FUNCTION_BLOCK FB_SFC_SamplePou
VAR_INPUT
//	eOperation	: INT;
	eOperation	: E_Operation;
END_VAR
VAR_OUTPUT
	iResultC	: DINT;
END_VAR
VAR
	arrDataA	: ARRAY [1..iMax] OF DINT;
	arrDataB	: ARRAY [1..iMax] OF DINT;
	arrDataC	: ARRAY [1..iMax] OF DINT;
	I 			: DINT;
	bInit		: BOOL := TRUE;
	bAdd		: BOOL;
	bSub		: BOOL;
	bMul		: BOOL;
END_VAR
VAR CONSTANT
	iMax 		: DINT := 10;
END_VAR

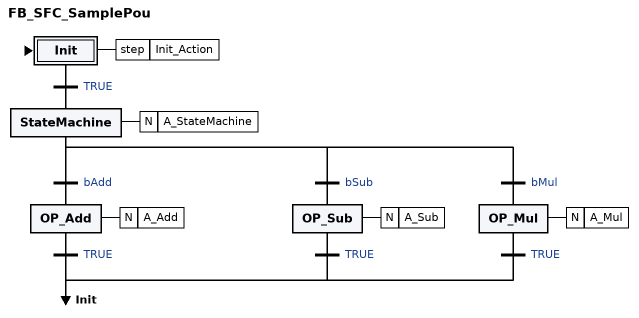
INITIAL_STEP Init:
    Init_Action(N);  // step action
END_STEP
TRANSITION FROM Init TO StateMachine
    := TRUE;
END_TRANSITION
STEP StateMachine:
    A_StateMachine(N);
END_STEP
TRANSITION FROM StateMachine TO OP_Add
    := bAdd;
END_TRANSITION
STEP OP_Add:
    A_Add(N);
END_STEP
TRANSITION FROM OP_Add TO Init
    := TRUE;
END_TRANSITION
TRANSITION FROM StateMachine TO OP_Sub
    := bSub;
END_TRANSITION
STEP OP_Sub:
    A_Sub(N);
END_STEP
TRANSITION FROM OP_Sub TO Init
    := TRUE;
END_TRANSITION
TRANSITION FROM StateMachine TO OP_Mul
    := bMul;
END_TRANSITION
STEP OP_Mul:
    A_Mul(N);
END_STEP
TRANSITION FROM OP_Mul TO Init
    := TRUE;
END_TRANSITION

ACTION A_Add:
(* WHILE - LOOP with check before first execution *)
iResultC := 0;
I := 1;
WHILE I <= iMax DO
	arrDataC[I] := arrDataA[I] + arrDataB[I];
	iResultC 	:= iResultC + arrDataC[I];
	I := I + 1;
END_WHILE
END_ACTION

ACTION A_Mul:
(* FOR - LOOP with check before first execution *)
iResultC := 1;
FOR I := 1 TO iMax DO
	arrDataC[I] := arrDataA[I] * arrDataB[I];
	iResultC 	:= iResultC * arrDataC[I];
END_FOR
END_ACTION

ACTION A_StateMachine:
bAdd := (eOperation = eOp_ADD);
bSub := (eOperation = eOp_SUB);
bMul := (eOperation = eOp_MUL);
END_ACTION

ACTION A_Sub:
(* REPEAT - LOOP: for array access *)
iResultC := 0;
I := 1;
REPEAT
	arrDataC[I] := arrDataA[I] - arrDataB[I];
	iResultC 	:= iResultC - arrDataC[I];
	I := I + 1;
UNTIL I > iMax END_REPEAT
END_ACTION

ACTION Init_Action:
IF bInit THEN
	bInit := FALSE;

	(* FOR loop: for array access *)
	FOR I := 1 TO iMax DO
		arrDataA[I] := I;
		arrDataB[I] := iMax - I + 1;
	END_FOR
END_IF
END_ACTION

END_FUNCTION_BLOCK

(* stored: Version 1.1.0.1, ProductVersion 3.1.4024.11
   POU FB_SFC_SamplePou: Id {6332420c-e0db-44ef-b583-644195b4910a}, SpecialFunc None
   Action A_Add: Id {52bd5163-7cab-4f97-b7c1-e81f980c20b5}
   Action A_Mul: Id {8a1edc83-bcc3-4c20-a7a8-cc9debe5ccd4}
   Action A_StateMachine: Id {69dacc95-257e-4e5a-b379-3a86d2b8ce55}
   Action A_Sub: Id {d0456552-6784-45ce-a35d-a7b70e42e6b0}
   Action Init_Action: Id {06469600-6efd-49eb-956c-9a6e1a063ef1} *)
